// TIA Portal V20 export
TYPE "LER_typeUnitHistory"
// stored: Access Published
   STRUCT
      hotPressLeft { ExternalWritable := 'False'; S7_SetPoint := 'True'} : "LER_typeServoPressHistory";
      hotPressRight { ExternalWritable := 'False'; S7_SetPoint := 'True'} : "LER_typeServoPressHistory";
      hipot { ExternalWritable := 'False'; S7_SetPoint := 'True'} : "LER_typeHipotHistory";
      thickness { ExternalWritable := 'False'; S7_SetPoint := 'True'} : "LER_typeThicknessHistory";
      vision { ExternalWritable := 'False'; S7_SetPoint := 'True'} : "LER_typeVisionHistory";
      laserMark { ExternalWritable := 'False'; S7_SetPoint := 'True'} : "LER_typeLaserMarkHistory";
      weightCheck { ExternalWritable := 'False'; S7_SetPoint := 'True'} : "LER_typeWeightCheckHistory";
   END_STRUCT;
END_TYPE
